PROGRAM MAIN
VAR
	bOut AT %Q*: ARRAY[0..7] OF BOOL;
	pwm AT %Q*: UINT;
	
END_VAR

pwm:=4000;

END_PROGRAM

(* stored: Version 1.1.0.1, ProductVersion 3.1.4024.4
   POU MAIN: Id {d2148b4f-ffc5-48fc-a830-0599cebfe4fc}, SpecialFunc None *)
